// TwinCAT 3 PLC project ModBus_Master_PLC
// ProgramVersion: 3.1.4023.0
// libraries:
//   Tc2_ModbusSrv, * (Beckhoff Automation GmbH)
//   Tc2_Standard, * (Beckhoff Automation GmbH)
//   Tc2_System, * (Beckhoff Automation GmbH)
//   Tc3_Module, * (Beckhoff Automation GmbH)
// project tree:
//   GVLs/ GVL.TcGVL
//   / PlcTask.TcTTO
//   POUs/ MAIN.TcPOU
// real-time tasks:
//   TASK PlcTask: cycle T#10ms, priority 20, ADS port 350

CONFIGURATION ModBus_Master_PLC
    RESOURCE PLC ON TwinCAT3
        TASK PlcTask(INTERVAL := T#10ms, PRIORITY := 20);
        PROGRAM MAIN WITH PlcTask : MAIN;
    END_RESOURCE
END_CONFIGURATION

// ---- GVLs/GVL.TcGVL
{attribute 'qualified_only'}
// These variable are mapped to the ModBus address ranges 0x8000 - 0x80FF for this device
VAR_GLOBAL
	mb_Input_Coils		: ARRAY[0..255] OF BOOL; // these coils can be queried by a MB master device using command 0x02
	mb_Output_Coils		: ARRAY[0..255] OF BOOL; // these coils can be set by a MB master device using 0x0f and queried by 0x01
	mb_Input_Registers	: ARRAY[0..255] OF WORD; // these registers are can be queried by a MB master device using command 0x04
	mb_Output_Registers	: ARRAY[0..255] OF WORD; // registers can be set by a MB device using 0x10, queried by 0x03 and 0x06
END_VAR

// ---- POUs/MAIN.TcPOU
PROGRAM MAIN
VAR

	bForceConfig	: BOOL;						// set this to re-run configuration for the MB FB
	sIpAdress		: STRING := '172.17.16.1';	// IP address of target device for ModBus functions

	// Write some random data to the other MODBUS slave 

	fb_MBWriteRegs	: FB_MBWriteRegs;

	fbSetRegTimer	: TON	:= (PT := T#2S);	// timer to set MB registers at certain interval 
	bStart			: BOOL;						// set this to set MB registers

	arrdata	 		: ARRAY[0..3] OF WORD;		// data to write to some MB registers
	uiRepeats		: UINT;						// number of times registers have been set
	iInt			: INT;						// iterator 
	

	// Set parameters for scrolling coils on other MODBUS device 

	fb_MBSetScroll	: FB_MBWriteSingleCoil;
	fb_MBWritePause	: FB_MBWriteSingleReg;

	bScroll			: BOOL;				// Set this to request the MB device scroll it's coils 
	uiPauseTime		: UINT	:= 500;		// Time in MS to pause between coils while scrolling
	
	// Internal to the scrolling logic
	bScrollPrev			: BOOL;	
	uiPauseTimePrev		: UINT;
	bTriggerScrollSet	: BOOL;
	bTriggerPauseSet	: BOOL;

END_VAR

// Set up MODBUS function blocks
IF(_TaskInfo[GETCURTASKINDEXEX()].FirstCycle OR bForceConfig) THEN
	bForceConfig			:= FALSE;
	
	// write registers - random data 
	fb_MBWriteRegs.sIPAddr	:= sIpAdress;
	fb_MBWriteRegs.nTCPPort	:= 502;
	fb_MBWriteRegs.nUnitID	:= 16#FF;			// set to 16#FF if addressing the target directly via TCP

	// write registers - control slave scroller 
	fb_MBWritePause.sIPAddr	:= sIpAdress;
	fb_MBWritePause.nTCPPort	:= 502;
	fb_MBWritePause.nUnitID	:= 16#FF;			// set to 16#FF if addressing the target directly via TCP
	
	// set coils 
	fb_MBSetScroll.sIPAddr	:= sIpAdress;
	fb_MBSetScroll.nTCPPort	:= 502;
	fb_MBSetScroll.nUnitID	:= 16#FF;			// set to 16#FF if addressing the target directly via TCP

END_IF





// Periodically write some data to MB registers 
fbSetRegTimer(IN:=TRUE);		// run our send update timer  
IF fbSetRegTimer.Q THEN			// if the timer has expired (its time to set the registers) 
	fbSetRegTimer(IN:=FALSE);  	// reset the timer 
	
	// Generate some new values for our registers
	FOR iInt:= 0 TO 3 BY 1 DO 
		arrData[iInt]	:= arrdata[iInt] + iInt + 1;	// increment each value by 1 
	END_FOR

	bStart		:= TRUE;					// start a new MODBUS set operation 
	uiRepeats	:= uiRepeats + 1;			// increment the repeats counter 
	
END_IF	

// Run the MB wite FB if requested and while still busy or in error 
IF(bStart OR fb_MBWriteRegs.bBusy OR fb_MBWriteRegs.bError) THEN	
		
	fb_MBWriteRegs(	nMBAddr		:= 16#8004, 
					nQuantity	:= 4, 
					cbLength	:= SIZEOF(arrdata), 
					pSrcAddr	:= ADR(arrdata), 
					bExecute	:= bStart, 
					tTimeout	:= T#2S, 
					bBusy=> , 
					bError=> , 
					nErrId=> );
					
	bStart	:= FALSE;	// reset the MB set start trigger 				
END_IF				

IF (bScroll <> bScrollPrev) THEN
	bTriggerScrollSet	:= TRUE;
END_IF

IF (uiPauseTime <> uiPauseTimePrev) THEN
	bTriggerPauseSet	:= TRUE;
END_IF
// Update the memory of the previous scroll pause value and scroll activation status 
bScrollPrev		:= bScroll;
uiPauseTimePrev	:= uiPauseTime;


// Run the MB setcoils FB if requested and while still busy or in error 
IF(bTriggerScrollSet OR fb_MBSetScroll.bBusy OR fb_MBSetScroll.bError) THEN	
	IF(bScroll) THEN	
		fb_MBSetScroll(	nMBAddr		:= 16#8000,
						nValue		:= 16#FF00,
						bExecute	:= bTriggerScrollSet,
						tTimeout	:= T#2S, 
						bBusy=> , 
						bError=> , 
						nErrId=> );
	ELSE
		fb_MBSetScroll(	nMBAddr		:= 16#8000,
						nValue		:= 16#0000,
						bExecute	:= bTriggerScrollSet,
						tTimeout	:= T#2S, 
						bBusy=> , 
						bError=> , 
						nErrId=> );
	END_IF					

	bTriggerScrollSet	:= FALSE;	// reset the MB set start trigger 				
END_IF				


// Run the MB setpause FB if requested and while still busy or in error 
IF(bTriggerPauseSet OR fb_MBWritePause.bBusy OR fb_MBWritePause.bError) THEN	
		
	fb_MBWritePause(nMBAddr		:= 16#8000, 
					nValue		:= UINT_TO_WORD(uiPauseTime),
					bExecute	:= bTriggerPauseSet, 
					tTimeout	:= T#2S, 
					bBusy=> , 
					bError=> , 
					nErrId=> );
					
	bTriggerPauseSet	:= FALSE;	// reset the MB set start trigger 				
END_IF

END_PROGRAM
